// TwinCAT 3 PLC project PLC_TMO_VAC_FS
// ProgramVersion: 3.1.4022.7
// libraries:
//   L2SI Vacuum Library, * (SLAC)
//   LCLS General, * (SLAC)
//   PMPS, * (SLAC - LCLS)
//   Tc2_Standard, * (Beckhoff Automation GmbH)
//   Tc2_System, * (Beckhoff Automation GmbH)
//   Tc3_Module, * (Beckhoff Automation GmbH)
// project tree:
//   / PlcTask.TcTTO
//   POUs/ MAIN.TcPOU
// (motion and I/O tree: see PLC project plc_tmo_vac)
// real-time tasks:
//   TASK PlcTask: cycle T#10ms, priority 20, ADS port 350
//   TASK ComTask: cycle T#11ms, priority 1, ADS port 351
//   TASK FSVTask: cycle T#2ms, priority 2, ADS port 352
// variable links:

CONFIGURATION PLC_TMO_VAC_FS
    RESOURCE PLC ON TwinCAT3
        TASK PlcTask(INTERVAL := T#10ms, PRIORITY := 20);
        PROGRAM MAIN WITH PlcTask : MAIN;
    END_RESOURCE
END_CONFIGURATION

// ---- POUs/MAIN.TcPOU
PROGRAM MAIN
VAR
	i_xFFReset: INT;
END_VAR

(*TV1K4_VFS_01(
	i_xPMPS_OK:= TRUE, 
	i_xExt_OK:= TRUE, 
	i_xOverrideMode:= FALSE, 
	iq_stValve=> );*)

END_PROGRAM
